# B&R Automation Studio project GroupProjectBR
Automation Studio 4.12.3.127 SP; Project that includes both HMI visualization and script of controling conveyor belt and sorting system.; technology packages: mapp 5.23.0, mappCockpit 5.23.0, mappMotion 5.23.0, mappView 5.23.0, mappVision 5.23.0

## Configuration ConfigSortingSystem

CPU , AutomationRuntime B4.93, Build 4.1.2, Safety 0.0, Vc V4.72.6

### Task classes (Cpu.sw)
```
Cyclic#4:
  Auto <- Programs.Auto.prg
  Camera <- Programs.Camera.prg
  Alarms <- Programs.Alarms.prg
  Manual <- Programs.Manual.prg
  ProgramRec <- Programs.RecipesMgmnt.prg
  SemiAuto <- Programs.SemiAuto.prg
DataObjects: McAcpSys
NcDataObjects: McDriveLog
Binaries: McAcpDrv, udbdef, McAcpSim, mvLoader, arflatprv, TCLang, visionUnit, mCoWebSc, TCData, FWRules, arcoal, arsvcreg, SettingsVi, sysconf, Settings, iomap, asfw, viComp, Role, ashwac, gRecipeXML, Config_2, arconfig, viAppLogo, Config_1, TC, ashwd, Config, User
Libraries: McBase, MpAxis, McAxis, MpBase, McAcpAx, CoTrace, AsZip, FileIO, runtime, ViBase, AsARCfg, powerlnk, MpRecipe, AsEPL, AsIO, DataObj, astime, MpAlarmX, MpServer, standard, AsHttp, asieccon, aruser, arssl, sys_lib, MpUserX
```

### Hardware
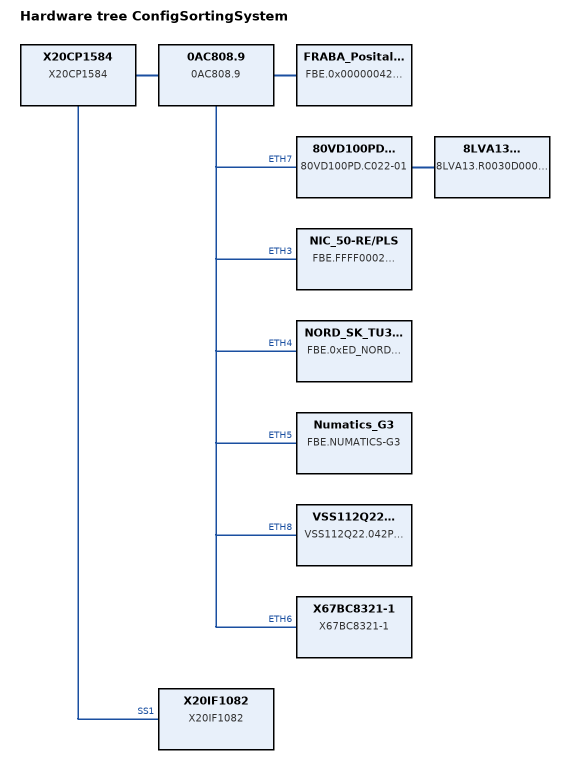
```
0AC808.9 : 0AC808.9 v1.0.0.0  [ETH1 -> X20CP1584.IF3 [Cable Type=PowerlinkCable, Length=10, Version=1.0.0.3]; ETH2 -> FRABA_Posital_Absolute_Rotary_Encoder.PLK1 [Cable Type=PowerlinkCable, Length=10, Version=1.0.0.3]; ETH3 -> NIC_50-RE/PLS.PLK1 [Cable Type=PowerlinkCable, Length=10, Version=1.0.0.3]; ETH4 -> NORD_SK_TU3-POL_SK54xE_Inverter.PLK1 [Cable Type=PowerlinkCable, Length=10, Version=1.0.0.3]; ETH5 -> Numatics_G3.PLK1 [Cable Type=PowerlinkCable, Length=10, Version=1.0.0.3]; ETH6 -> X67BC8321-1.PLK1 [Cable Type=PowerlinkCable, Length=10, Version=1.0.0.3]; ETH7 -> 80VD100PD.C022-01.PLK2 [Cable Type=PowerlinkCable, Length=10, Version=1.0.0.3]; ETH8 -> VSS112Q22.042P-000.PLK1 [Cable Type=PowerlinkCable, Length=10, Version=1.0.0.3]]
80VD100PD.C022-01 : 80VD100PD.C022-01 v2.5.0.0  [PLK2 -> 0AC808.9.ETH7 (NodeNumber=9) [Cable Type=PowerlinkCable, Length=10, Version=1.0.0.3]]
  DriveConfiguration/Module:
    McAcoposTypeID = AcoposMicroDConfig
    ActivateACOPOSSimulationOnPLC = 0
  DriveConfiguration/Encoder/EncoderX6A/InterfaceType:
    ResolverPolepairs = 1
  DriveConfiguration/Encoder/EncoderX6B/InterfaceType:
    ResolverPolepairs = 1
  DriveConfiguration/Channel[1]/RealAxis:
    AxisReference = gAxis_1
    MechanicalElementsIsInvisible = 0
  DriveConfiguration/Channel[1]/RealAxis/MechanicalElements/Gearbox:
    InputIsReadOnly = 0
    Input = 1
    OutputIsReadOnly = 0
    Output = 1
  DriveConfiguration/Channel[1]/RealAxis/MechanicalElements/RotaryToLinearTransformation:
    ReferenceDistanceIsReadOnly = 0
    ReferenceDistance = 175
  DriveConfiguration/Channel[1]/RealAxis/Controller:
    ModeIsReadOnly = 0
    Mode = PositionController
  DriveConfiguration/Channel[1]/RealAxis/Controller/Mode/Position:
    ProportionalGain = 194
    IntegrationTime = 0.0
    PredictionTime = 0.0004
    TotalDelayTime = 0.0004
  DriveConfiguration/Channel[1]/RealAxis/Controller/Mode/Speed:
    ProportionalGainIsReadOnly = 0
    ProportionalGain = 0.75
    IntegrationTimeIsReadOnly = 0
    IntegrationTime = 0.0
    FilterTimeIsReadOnly = 0
    FilterTime = 0.0
  DriveConfiguration/Channel[1]/RealAxis/Controller/Mode/LoopFilters:
    LoopFilterXIsReadOnly = 0
    LoopFilter1 = NotUsed
    LoopFilter2 = NotUsed
    LoopFilter3 = NotUsed
  DriveConfiguration/Channel[1]/RealAxis/Homing:
    ModeIsReadOnly = 0
    Mode = Direct
  DriveConfiguration/Channel[1]/RealAxis/Homing/Mode:
    Position = 0.0
    ReferencePulse = NotUsed
  DriveConfiguration/Channel[1]/RealAxis/Homing:
    RestorePositionVariable = 
  DriveConfiguration/Channel[1]/RealAxis/StopReaction:
    QuickstopIsReadOnly = 0
    Quickstop = DecelerationLimit
    DriveErrorIsReadOnly = 0
    DriveError = DecelerationLimit
  DriveConfiguration/Channel[1]/RealAxis/MovementErrorLimits:
    PositionError = 5
    VelocityErrorMonitoring = Automatic1
  DriveConfiguration/Channel[1]/RealAxis:
    JerkFilterIsReadOnly = 0
    JerkFilter = NotUsed
    ZeroVibrationFilter = NotUsed
  DriveConfiguration/Channel[1]/RealAxis/DigitalInputs/HomingSwitch:
    SourceIsReadOnly = 0
    Source = NotUsed
    Level = High
  DriveConfiguration/Channel[1]/RealAxis/DigitalInputs/PositiveLimitSwitch:
    SourceIsReadOnly = 0
    Source = NotUsed
    Level = High
  DriveConfiguration/Channel[1]/RealAxis/DigitalInputs/NegativeLimitSwitch:
    SourceIsReadOnly = 0
    Source = NotUsed
    Level = High
  DriveConfiguration/Channel[1]/RealAxis/DigitalInputs/Trigger1:
    Source = X2Trigger1
    Level = High
  DriveConfiguration/Channel[1]/RealAxis/DigitalInputs/Trigger2:
    Source = X2Trigger2
    Level = High
  DriveConfiguration/Channel[1]/RealAxis/DigitalInputs/Quickstop:
    Input = Trigger2
  DriveConfiguration/Channel[1]/RealAxis/Simulation:
    SimulationModeOnPLC = SetValueGeneration
    SimulationModeOnACOPOS = NotUsed
  DriveConfiguration/Channel[2]/RealAxis:
    AxisReference = 
    MechanicalElementsIsInvisible = 0
  DriveConfiguration/Channel[2]/RealAxis/MechanicalElements/Gearbox:
    InputIsReadOnly = 0
    Input = 1
    OutputIsReadOnly = 0
    Output = 1
  DriveConfiguration/Channel[2]/RealAxis/MechanicalElements/RotaryToLinearTransformation:
    ReferenceDistanceIsReadOnly = 0
    ReferenceDistance = 1
  DriveConfiguration/Channel[2]/RealAxis/Controller:
    ModeIsReadOnly = 0
    Mode = PositionController
  DriveConfiguration/Channel[2]/RealAxis/Controller/Mode/Position:
    ProportionalGain = 50.0
    IntegrationTime = 0.0
    PredictionTime = 0.0004
    TotalDelayTime = 0.0004
  DriveConfiguration/Channel[2]/RealAxis/Controller/Mode/Speed:
    ProportionalGainIsReadOnly = 0
    ProportionalGain = 2.0
    IntegrationTimeIsReadOnly = 0
    IntegrationTime = 0.0
    FilterTimeIsReadOnly = 0
    FilterTime = 0.0
  DriveConfiguration/Channel[2]/RealAxis/Controller/Mode/LoopFilters:
    LoopFilterXIsReadOnly = 0
    LoopFilter1 = NotUsed
    LoopFilter2 = NotUsed
    LoopFilter3 = NotUsed
  DriveConfiguration/Channel[2]/RealAxis/Homing:
    ModeIsReadOnly = 0
    Mode = Direct
  DriveConfiguration/Channel[2]/RealAxis/Homing/Mode:
    Position = 0.0
    ReferencePulse = NotUsed
  DriveConfiguration/Channel[2]/RealAxis/Homing:
    RestorePositionVariable = 
  DriveConfiguration/Channel[2]/RealAxis/StopReaction:
    QuickstopIsReadOnly = 0
    Quickstop = DecelerationLimit
    DriveErrorIsReadOnly = 0
    DriveError = DecelerationLimit
  DriveConfiguration/Channel[2]/RealAxis/MovementErrorLimits:
    PositionError = 1.0
    VelocityErrorMonitoring = Automatic1
  DriveConfiguration/Channel[2]/RealAxis:
    JerkFilterIsReadOnly = 0
    JerkFilter = NotUsed
    ZeroVibrationFilter = NotUsed
  DriveConfiguration/Channel[2]/RealAxis/DigitalInputs/HomingSwitch:
    SourceIsReadOnly = 0
    Source = NotUsed
    Level = High
  DriveConfiguration/Channel[2]/RealAxis/DigitalInputs/PositiveLimitSwitch:
    SourceIsReadOnly = 0
    Source = NotUsed
    Level = High
  DriveConfiguration/Channel[2]/RealAxis/DigitalInputs/NegativeLimitSwitch:
    SourceIsReadOnly = 0
    Source = NotUsed
    Level = High
  DriveConfiguration/Channel[2]/RealAxis/DigitalInputs/Trigger1:
    Source = X2Trigger1
    Level = High
  DriveConfiguration/Channel[2]/RealAxis/DigitalInputs/Trigger2:
    Source = X2Trigger2
    Level = High
  DriveConfiguration/Channel[2]/RealAxis/DigitalInputs/Quickstop:
    Input = Trigger2
  DriveConfiguration/Channel[2]/RealAxis/Simulation:
    SimulationModeOnPLC = SetValueGeneration
    SimulationModeOnACOPOS = NotUsed
8LVA13.R0030D000-0 : 8LVA13.R0030D000-0 v2.2.0.4  [MT -> 80VD100PD.C022-01.MT1]
  M1/MotorParameters:
    MOTOR_AMB_TEMP_RATED = 40
FRABA_Posital_Absolute_Rotary_Encoder : FBE.0x00000042_PowerlinkRotaryEncoder_OCD_V02-10 v1.0 (OrderNumber=FRABA Posital Absolute Rotary Encoder)  [PLK1 -> 0AC808.9.ETH2 (NodeNumber=8) [Cable Type=PowerlinkCable, Length=10, Version=1.0.0.3]]
  Supervision = off
  p2110_value = 
  p6000_value = 
  p6003_value = 
NIC_50-RE/PLS : FBE.FFFF0002_TLBPOWERLINK v1.0 (OrderNumber=NIC 50-RE/PLS)  [PLK1 -> 0AC808.9.ETH3 (NodeNumber=2) [Cable Type=PowerlinkCable, Length=10, Version=1.0.0.3]]
  Supervision = off
NORD_SK_TU3-POL_SK54xE_Inverter : FBE.0xED_NORD_TU3_POL_SK54xE_Inverter v1.0 (OrderNumber=NORD SK TU3-POL SK54xE Inverter)  [PLK1 -> 0AC808.9.ETH4 (NodeNumber=3) [Cable Type=PowerlinkCable, Length=10, Version=1.0.0.3]]
  Supervision = off
Numatics_G3 : FBE.NUMATICS-G3 v1.0 (OrderNumber=Numatics G3)  [PLK1 -> 0AC808.9.ETH5 (NodeNumber=6) [Cable Type=PowerlinkCable, Length=10, Version=1.0.0.3]]
  Supervision = off
VSS112Q22.042P-000 : VSS112Q22.042P-000 v1.7.0.605  [PLK1 -> 0AC808.9.ETH8 (NodeNumber=1) [Cable Type=PowerlinkCable, Length=10, Version=1.0.0.3]]
  Supervision = off
  VisionConfig = gCamera
X20CP1584 : X20CP1584 v1.10.0.0
  Connector IF2:
    ActivateDevice = 1
    Mode = Manual
    InternetAddress = 192.168.0.100
    SubnetMask = 255.255.255.0
    ActivateSnmp = 2
  Connector IF3:
    MtuSize = 1500
    CycleTime = 400
    InternetAddress = 192.168.200.240
    SubnetMask = 255.255.255.0
    ActivateANSL = 1
  ConfigurationID = Group_Project_BR_ConfigSortingSystem
  Simulation = 1
  TimerDeviceType = EPLX2X
  TimerDevice = X20CP1584.IF3
  TaskClassIdleTime = 2000
  FileDevice1
  FileDeviceName1 = CF
  FileDevicePath1 = C:\Users\Szkolenie\Desktop\Recipies
  FileDevice2
  FileDeviceName2 = TegesSmeges
  FileDevicePath2 = C:\Users\barto\OneDrive\Pulpit\Folder na receptury
  TimeZone = 160
  ActivateDaylightSavingTime = 1
  ActivateOpcUa = 1
  OpcUaInformationModels_PV_Version = 1
X20IF1082 : X20IF1082 v1.12.0.0  [SS -> X20CP1584.SS1]
  Connector IF1:
    EplNatSubnet = 192.168.102.0
X67BC8321-1 : X67BC8321-1 v2.14.0.0  [PLK1 -> 0AC808.9.ETH6 (NodeNumber=5) [Cable Type=PowerlinkCable, Length=10, Version=1.0.0.3]]
```

### IoMap.iom - X20CP1584/IoMap.iom
```iecst
VAR_CONFIG
	::gInWeightMeasure AT %IB."NIC_50-RE/PLS"._1ByteIn_04_I2100_S04;
	::Camera:PhotosTaken AT %IB."VSS112Q22.042P-000".CompletedAcquisitionCnt;
	::gActuatorByte AT %QW."Numatics_G3".Out01_I3201Out;
	::gImageAcq AT %QX."VSS112Q22.042P-000".ImageAcquisition;
	::Camera:SET_FOCUS AT %QW."VSS112Q22.042P-000".SetFocus;
	::Camera:EXPO_TIME AT %QD."VSS112Q22.042P-000".ExposureTime01;
	::Camera:NumberMatches AT %IB."VSS112Q22.042P-000".NumResultsMatch;
	::Camera:RecognisedModel AT %IB."VSS112Q22.042P-000".ModelNumberMatch01;
	::Camera:MatchEnable AT %QX."VSS112Q22.042P-000".EnableMatch;
	::Camera:NUM_SEARCH_MAX AT %QB."VSS112Q22.042P-000".NumSearchMaxMatch;
	::Camera:MIN_SCORE AT %QB."VSS112Q22.042P-000".MinScoreMatch;
	::Camera:MAX_OVERLAP AT %QB."VSS112Q22.042P-000".MaxOverlapMatch;
	::Camera:FLASH_COLOR AT %QB."VSS112Q22.042P-000".FlashColor01;
	::Camera:FLASH_SEGMENT AT %QB."VSS112Q22.042P-000".FlashSegment01;
	::Camera:MatchScore AT %IB."VSS112Q22.042P-000".ScoreMatch01;
	::Camera:CameraLED_OPC AT %QB."VSS112Q22.042P-000".StatusLED;
	::Camera:ImgProcessingActive AT %IX."VSS112Q22.042P-000".ImageProcessingActive;
	::Alarms:ModuleOkCamera AT %IX."VSS112Q22.042P-000".ModuleOk;
	::Alarms:ModuleOkScale AT %IX."NIC_50-RE/PLS".ModuleOk;
	::Alarms:ModuleOkInverter AT %IX."NORD_SK_TU3-POL_SK54xE_Inverter".ModuleOk;
	::Alarms:ModuleOkPLC_PLK AT %IX."X20IF1082".ModuleOk;
	::Alarms:ModuleOkEncoder AT %IX."FRABA_Posital_Absolute_Rotary_Encoder".ModuleOk;
	::Alarms:ModuleOkActuators AT %IX."Numatics_G3".ModuleOk;
	::Alarms:ModuleOkPneu_X67BC AT %IX."X67BC8321-1".ModuleOk;
END_VAR
```

### Config.mpalarmxcore - X20CP1584/mappServices/Config.mpalarmxcore
```
Element gAlarmXCore (Type=mpalarmxcore)
  mapp.AlarmX.Core.Configuration:
    [0]:
      Name = Unrecognized object
      Message = Attempt to classify object has failed
      Behavior = DiscreteValueMonitoring
        Monitoring:
          MonitoredPV = ::Auto:State
          TriggerValues:
            [0] = 14
    [1]:
      Name = Left box is full
      Message = Left box reached maximum ammount of objects in it
      Behavior = LevelMonitoring
        Monitoring:
          MonitoredPV = ::Auto:QuantityLeftStorage
          HighLimitEnable = Dynamic
            LimitPV = ::gMaxLeftStorage
    [2]:
      Name = Right box is full
      Message = Right box reached maximum ammount of objects in it
      Behavior = LevelMonitoring
        Monitoring:
          MonitoredPV = ::Auto:QuantityRightStorage
          HighLimitEnable = Dynamic
            LimitPV = ::gMaxRightStorage
    [3]:
      Name = Motor error
      Message = gMotorBeltAxisBasic has returned an error. Manual restart is required in "Service" page.
      Behavior = DiscreteValueMonitoring
        Monitoring:
          MonitoredPV = ::gMotorBeltAxisBasic.Error
          TriggerValues:
            [0] = 1
    [4]:
      Name = Right box is full (manual)
      Message = Right box reached maximum ammount of objects in it (manual mode)
      Behavior = LevelMonitoring
        Monitoring:
          MonitoredPV = ::SemiAuto:QuantityRightStorage
          HighLimitEnable = Dynamic
            LimitPV = ::gMaxRightStorage
    [5]:
      Name = Left box is full (manual)
      Message = Left box reached maximum ammount of objects in it (manual mode)
      Behavior = LevelMonitoring
        Monitoring:
          MonitoredPV = ::SemiAuto:QuantityLeftStorage
          HighLimitEnable = Dynamic
            LimitPV = ::gMaxRightStorage
    [6]:
      Name = Hardware error
      Message = No connection to at least on module. Fix connections and reset hardware via service page
      Behavior = DiscreteValueMonitoring
        Monitoring:
          MonitoredPV = ::gAlarmHardware
          TriggerValues:
            [0] = 1
```

### viComp.visioncomponent - X20CP1584/mappVision/viComp.visioncomponent
```
Element gCamera (Type=visioncomponent)
  VisionApplicationReference = viAppLogo
```

## Logical view

Binary libraries used (declarations not repeated): operator, runtime, astime, AsIecCon, MpAxis, McAxis, MpBase, McAcpAx, CoTrace, AsZip, FileIO, McBase, MpRecipe, asstring, ViBase, AsARCfg, powerlnk, AsEPL, AsIO, DataObj, MpAlarmX, MpServer, standard, AsHttp

### Global.typ - Global data types
```iecst
TYPE
	ModelEnum :
		(
		BR := 1, (*%ID of B&R logo model*)
		AS := 2, (*%ID of AS logo model*)
		Unrecognised := 0 (*%case of nothing recognised*)
		);
	CofeeType : 	STRUCT
		Sugar : USINT;
		Water : REAL;
		Powder : USINT;
		Temperature : REAL;
		Milk : REAL;
	END_STRUCT;
	SortingType : 	STRUCT
		RecognisedModel : ModelEnum; (*Model rozpoznany*)
		ItemWeightChoosen : USINT := 10;
		SortLeftMin : BOOL := FALSE; (*Mniejsze detale sortowane są na lewo gdy 1, a wieksze na prawo gdy 1.*)
		SortLeftBR : BOOL := FALSE; (*Gdy ustawiona na 1 sortuje BR na lewo, a AS na prawo*)
		SortChoice : SortChoiceEnum;
	END_STRUCT;
	SortChoiceEnum :
		(
		WEIGHT,
		OPTIC
		);
END_TYPE
```

### Global.var - Global variables
```iecst
(*Insert your comment here.*)
VAR
	Coffee : CofeeType;
	gActuatorByte : UINT;
	gAlarmExist : BOOL := FALSE;
	gAlarmHardAck : BOOL := FALSE;
	gAlarmHardware : BOOL := FALSE;
	gAutoRecipe : USINT;
	gErrorState : BOOL := FALSE;
	gExposureTime : UDINT;
	gImageAcq : BOOL := FALSE; (*Enabling image acquisition therefore starting matching procedure, rising edge*)
	gInWeightMeasure : USINT;
	gItemWeightChoosen : USINT := 10;
	gMaxLeftStorage : USINT := 4;
	gMaxRightStorage : USINT := 4;
	gMode : USINT := 0;
	gMotorBeltAxisBasic : MpAxisBasic;
	gMotorBeltParType : MpAxisBasicParType;
	gMpRecipeRegPar_0 : MpRecipeRegPar;
	gMpRecipeUI_0 : MpRecipeUI;
	gMpRecipeXML_0 : MpRecipeXml;
	gPicNotRecognised : BOOL := FALSE;
	gRecognisedModel : ModelEnum := Unrecognised; (*Value showing recognised model 1- B&R, 2- AS, 0- not recognised*)
	gSetFocus : USINT;
	gSortChoice : SortChoiceEnum := WEIGHT;
	gSortChoiceView : BOOL;
	gSorting : SortingType;
	gStopBlink : BOOL := TRUE;
	gStopState : BOOL := TRUE;
	gUIConnect : MpRecipeUIConnectType;
	gUISetup : MpRecipeUISetupType;
	gWeightDetected : BOOL := FALSE;
	gDisplayImg : BOOL;
END_VAR
```

### Package Logical/Libraries - Global libraries

- Visualisation Logical/mappView (not shown)

### Program Logical/Programs/Auto (IEC)

#### Types.typ
```iecst
TYPE
	ProgramStatesEnum :
		(
		STOP,
		INIT,
		DETECTION,
		CATEGORIZATION,
		SORT_STORAGE_LEFT,
		SORT_STORAGE_RIGHT,
		SORT_WEIGHT,
		SORT_WEIGHT_AND_OPTIC,
		SORT_OPTIC,
		STOP_AND_MANUAL,
		GO_STORAGE_LEFT,
		GO_STORAGE_RIGHT,
		TAKE_PICT_CAMERA,
		DROP,
		UNRECOGNISED_PIC,
		ERROR
		);
END_TYPE
```

#### Variables.var
```iecst
VAR
	TIME_TON_DETECT : TIME := T#2S;
END_VAR
VAR CONSTANT
	TIME_TON_CAMERA : TIME := T#4S;
	TIME_TON_ACTUATOR : TIME := T#500MS;
END_VAR
VAR
	TimerTonDetect : TON;
	TimerTonCamera : TON;
	TimerTonActuatorIn : BOOL := FALSE;
	TimerTonActuator : TON;
	TimerCameraPicDone : BOOL;
	TimerAfterDetect : BOOL;
	TimerActuatorOut : BOOL;
	StringState : STRING[80];
	StringRecognisedModel : STRING[80];
	Stop : BOOL := FALSE;
	State : ProgramStatesEnum := STOP;
	Start : BOOL := FALSE;
	SelectedAuto : BOOL;
	RESET_ITEM_MEM_WEIGHT : {REDUND_UNREPLICABLE} USINT := 0;
	NotSelectedAuto : BOOL;
END_VAR
VAR CONSTANT
	MOTOR_DIST_RIGHT : UINT := 320;
	MOTOR_DIST_LEFT : UINT := 90;
END_VAR
VAR
	MotorVel : REAL;
	MotorResetError : BOOL := FALSE;
	MotorReqVel : {REDUND_UNREPLICABLE} UINT := 300;
	MotorReqPosition : UINT := 0;
	MotorReqDec : UINT := 700;
	MotorReqAcc : UINT := 700;
	MotorPower : BOOL := FALSE;
	MotorPos : LREAL;
	MotorMoveDone : BOOL;
	MotorMoveAbsolute : BOOL := FALSE;
	MotorInPosition : BOOL;
	MotorHome : BOOL;
	ItemWeightMeasured : USINT;
	ItemWeight : USINT;
	ItemDetected : BOOL := FALSE;
	IsEnglishSelected : BOOL := TRUE;
END_VAR
VAR CONSTANT
	ACTUATOR_BYTE_SORT : INT := 2#0000000000000001;
	ACTUATOR_BYTE_PUSH : INT := 2#0000000000000100;
	ACTUATOR_BYTE_NOT_ACTIV : USINT := 2#0000000000000000;
END_VAR
VAR
	ActuatorSorting : BOOL := FALSE;
	ActuatorPushing : BOOL := FALSE;
	ActuatorNotSorting : BOOL;
	ActuatorNotPushing : BOOL;
	ActuatorByte : INT := 2#0000000000000000;
END_VAR
```

#### Main.st
```iecst
PROGRAM _INIT
	// NEED ONLY FOR WATCH
	gAxis_1;
	gMotorBeltParType;
	gMotorBeltAxisBasic;
END_PROGRAM
//po namyśle można było użyć struktur do zmiennych :P
PROGRAM _CYCLIC

	SelectedAuto := (gMode = 0);
	NotSelectedAuto := NOT SelectedAuto;

	// CODE WORKS ONLY WHEN AUTO IS ACTIVE
	IF  SelectedAuto THEN
		// MOTOR MANAGEMENT
		gMotorBeltAxisBasic.Enable 		:= TRUE;
		gMotorBeltAxisBasic.MpLink 		:= ADR(gAxis_1);
		gMotorBeltAxisBasic.Parameters 	:= ADR(gMotorBeltParType);
		MotorMoveDone 					:= gMotorBeltAxisBasic.MoveDone;
		gMotorBeltAxisBasic.Power 		:= MotorPower;
		gMotorBeltAxisBasic.Home 		:= MotorHome;

		gMotorBeltAxisBasic();

		// IN STATE STOP VALUES DOESN'T FLUCTUATE
		IF gMotorBeltAxisBasic.Velocity > 15 THEN
			MotorVel := gMotorBeltAxisBasic.Velocity;
		ELSE
			MotorVel := 0;
		END_IF;
		IF gMotorBeltAxisBasic.Position > 5 THEN
			MotorPos := gMotorBeltAxisBasic.Position;
		ELSE
			MotorPos := 0;
		END_IF;

		// ASSIGNING MOTION PARAMETERS
		gMotorBeltParType.Acceleration 	:= MotorReqAcc;
		gMotorBeltParType.Deceleration 	:= MotorReqDec;
		gMotorBeltParType.Velocity 		:= MotorReqVel;
		gMotorBeltParType.Position 		:= MotorReqPosition;

		// ASSIGNING GLOBAL VARIABLES TO LOCAL VARIABLES
		gActuatorByte					 := ActuatorByte;
		gMotorBeltAxisBasic.Power 		 := MotorPower;
		gMotorBeltAxisBasic.MoveAbsolute := MotorMoveAbsolute;
		gStopState 						 := (State = 0);

		// ASSIGNING LOCAL VARIABLES TO GLOBAL VARIABLES
		MotorInPosition 				 := gMotorBeltAxisBasic.InPosition;
		ItemWeight 						 := gInWeightMeasure;

		// ITEM DETECTION CONDITION
		ItemDetected := (ItemWeight > 1);
		gWeightDetected := ItemDetected;

		// TIMERS
		// actuator
		TimerTonActuator(IN := TimerTonActuatorIn, PT := TIME_TON_ACTUATOR);
		TimerActuatorOut := TimerTonActuator.Q;
		// camera
		TimerTonCamera(IN := gImageAcq , PT := TIME_TON_CAMERA);
		TimerCameraPicDone := TimerTonCamera.Q;
		// delay after detection
		TimerTonDetect.IN := ItemDetected;
		TimerTonDetect.PT := TIME_TON_DETECT;
		TimerAfterDetect := TimerTonDetect.Q;
		TimerTonDetect();

	END_IF;

	// ALARM OR STOP OR AUTO NOT ACTIVE
	IF	gAlarmHardware THEN
		IF NOT (State = ERROR) THEN
			State := ERROR;
		END_IF;
	ELSIF Stop OR gMode <> 0 OR gAlarmExist THEN
		Stop := FALSE;
		State := STOP;
	END_IF;

	// PROGRAM AUTO
	CASE State OF
		STOP:
			IF SelectedAuto THEN
				MotorPower 		  := FALSE;
				MotorMoveAbsolute := FALSE;
				MotorHome 		  := FALSE;
			END_IF;
			MotorPos := 0;
			MotorVel := 0;
			StringState := 'Stop';
			TimerTonActuatorIn 	  := FALSE;
			ActuatorSorting 	  := FALSE;
			ActuatorPushing  	  := FALSE;
			IF Start THEN
				State := INIT;
			END_IF;

		INIT:
			StringState 		:= 'Inicjalizacja';
			gAddToRight 		:= FALSE;
			gAddToLeft 			:= FALSE;
			TimerTonActuatorIn 	:= FALSE;
			ActuatorSorting 	:= FALSE;
			ActuatorPushing 	:= FALSE;
			MotorMoveAbsolute 	:= FALSE;
			MotorPower 			:= TRUE;
			MotorHome 			:= TRUE;
			gPicNotRecognised	:= FALSE;
			State 				:= START;

		START:
			StringState 		:= 'Gotowy do startu';
			IF ItemDetected THEN
				ItemWeightMeasured 	:= RESET_ITEM_MEM_WEIGHT;
				State := DETECTION;
			END_IF;

		DETECTION:
			MotorHome 	:= FALSE;
			StringState := 'Wykrycie detalu';
			IF TimerAfterDetect THEN
				ItemWeightMeasured := ItemWeight;
				State := CATEGORIZATION;
			END_IF;

		CATEGORIZATION:
			StringState := 'Kategoryzacja detalu';
			IF gSorting.SortChoice = WEIGHT THEN
				State := DROP;
			ELSIF gSorting.SortChoice = OPTIC THEN
				State := TAKE_PICT_CAMERA;
			END_IF;

		TAKE_PICT_CAMERA:
			StringState := 'Robienie zdjecia';
			gImageAcq 	:= TRUE;
			IF TimerCameraPicDone THEN
				gDisplayImg := TRUE;
				IF gSorting.RecognisedModel = 0 THEN 						//0
					gImageAcq 			  := FALSE;
					StringRecognisedModel := 'Unrecognised';
					State 				  := UNRECOGNISED_PIC;
				ELSE
					State 				  := DROP;
				END_IF;
			END_IF;

		DROP:
			StringState := 'Dozowanie detalu';
			ActuatorPushing := TRUE;
			IF TimerActuatorOut THEN
				ActuatorPushing := FALSE;
				IF gSorting.SortChoice = OPTIC THEN
					gSortChoiceView := TRUE;
					State := SORT_OPTIC;
				ELSIF gSorting.SortChoice = WEIGHT THEN
					gSortChoiceView := FALSE;
					State := SORT_WEIGHT;
				END_IF;
			END_IF;

			// ABOVE 1 TO ItemWeightChoosen ITEM FALL INTO THE LEFT, EQUAL AND ABOVE ItemWeightChoosen INTO THE RIGHT
		SORT_WEIGHT:
			StringState := 'Sortowanie wagowe';
			IF ItemWeightMeasured > 1 AND ItemWeightMeasured < gSorting.ItemWeightChoosen THEN
				IF gSorting.SortLeftMin THEN
					State := GO_STORAGE_LEFT;
				ELSE
					State := GO_STORAGE_RIGHT;
				END_IF;
			ELSIF ItemWeightMeasured >= gSorting.ItemWeightChoosen THEN
				IF gSorting.SortLeftMin THEN
					State := GO_STORAGE_RIGHT;
				ELSE
					State := GO_STORAGE_LEFT;
				END_IF;
			END_IF;

		SORT_OPTIC:
			StringState := 'Sortowanie optyczne';
			IF gSorting.RecognisedModel = 1 THEN
				gImageAcq 			  := FALSE;
				StringRecognisedModel := 'B&R';							//1
				IF gSorting.SortLeftBR THEN
					State := GO_STORAGE_LEFT;
				ELSE
					State := GO_STORAGE_RIGHT;
				END_IF;

			ELSIF gSorting.RecognisedModel = 2 THEN
				gImageAcq 			  := FALSE;
				StringRecognisedModel := 'AS';							//2
				IF gSorting.SortLeftBR THEN
					State := GO_STORAGE_RIGHT;
				ELSE
					State := GO_STORAGE_LEFT;
				END_IF;
			END_IF;

		GO_STORAGE_LEFT:
			StringState := 'Transport detalu do lewego zbiornika';
			MotorReqPosition := MOTOR_DIST_LEFT;
			MotorMoveAbsolute := TRUE;
			IF MotorInPosition AND MotorMoveDone THEN
				State := SORT_STORAGE_LEFT;
			END_IF;

		GO_STORAGE_RIGHT:
			StringState := 'Transport detalu do prawego zbiornika';
			MotorReqPosition  := MOTOR_DIST_RIGHT;
			MotorMoveAbsolute := TRUE;
			IF MotorInPosition AND MotorMoveDone THEN
				State := SORT_STORAGE_RIGHT;
			END_IF;

		SORT_STORAGE_LEFT:
			StringState := 'Zepchniecie detalu z tasmy do zbiornika lewego';
			MotorMoveAbsolute := FALSE;
			ActuatorSorting   := TRUE;
			gAddToLeft 		  := TRUE;
			IF TimerActuatorOut THEN
				State := INIT;
			END_IF;

		SORT_STORAGE_RIGHT:
			gAddToRight := TRUE;
			MotorMoveAbsolute := FALSE;
			State := INIT;

		UNRECOGNISED_PIC:
			StringState := 'Nie rozpoznano zdjecia';
			gPicNotRecognised := TRUE;
			State := STOP;

		ERROR: // SPONTANICZNA DECYZJA CTRL V Z STOP DLA LEPSZEJ FUNKCJONALNOŚCI - BRAKLO CZASU NA DOKLADNIEJSZE POPRAWKI
			IF gMode = 0 THEN
				MotorPower 		  := FALSE;
				MotorMoveAbsolute := FALSE;
				MotorHome 		  := FALSE;
			END_IF;
			MotorPos := 0;
			MotorVel := 0;
			TimerTonActuatorIn 	  := FALSE;
			ActuatorSorting 	  := FALSE;
			ActuatorPushing  	  := FALSE;
			StringState := 'Wystapil blad';
			gErrorState := TRUE;
			IF gAlarmHardAck THEN
				IF NOT gAlarmHardware THEN
					gAlarmHardAck := FALSE;
					gErrorState := FALSE;
					State := STOP;
				END_IF;
			END_IF;

	END_CASE;

	// TIMER INPUT TRIGGER TO DELAY ACTUATORS
	IF ActuatorPushing OR ActuatorSorting THEN
		TimerTonActuatorIn := TRUE;
	ELSE
		TimerTonActuatorIn := FALSE;
	END_IF;

	// OPERATION OF BYTE ACTUATORS WITH TIMER
	IF ActuatorPushing THEN
		ActuatorByte := ACTUATOR_BYTE_PUSH;
		IF TimerActuatorOut THEN
			ActuatorPushing := FALSE;
		END_IF;
	ELSIF ActuatorSorting THEN
		ActuatorByte := ACTUATOR_BYTE_SORT;
		IF TimerActuatorOut THEN
			ActuatorSorting := FALSE;
		END_IF;
	ELSE
		ActuatorByte := ACTUATOR_BYTE_NOT_ACTIV;
	END_IF;

	// COUNTERS
	gCTU_QuantityLeft(CU := gAddToLeft, RESET := gCTU_Reset_Left, PV := gMaxLeftStorage);
	gCTU_QuantityRight(CU := gAddToRight, RESET := gCTU_Reset_Right, PV := gMaxRightStorage);
	gQuantityLeftStorage  := gCTU_QuantityLeft.CV;
	gQuantityRightStorage := gCTU_QuantityRight.CV;

	gCTU_QuantityLeft();
	gCTU_QuantityRight();

	// HMI GUYS WANTED SOME VARIABLES
	IF gSorting.SortChoice = OPTIC THEN
		gSortChoiceView := TRUE;
	ELSIF gSorting.SortChoice = WEIGHT THEN
		gSortChoiceView := FALSE;
	END_IF;

	ActuatorNotSorting := NOT ActuatorSorting;
	ActuatorNotPushing 	:= NOT ActuatorPushing;

	IF Start THEN
		Start := FALSE;
	END_IF;

	//Added by Jakub; Responsibler for changing machine state between English and Polish
	IF IsEnglishSelected THEN
		IF StringState = 'Inicjalizacja' THEN
			StringState := 'Initialization';

		ELSIF StringState = 'Gotowy do startu' THEN
			StringState := 'Ready';

		ELSIF StringState = 'Wykrycie detalu' THEN
			StringState := 'Item detection';

		ELSIF StringState = 'Kategoryzacja detalu' THEN
			StringState := 'Item categorization';

		ELSIF StringState = 'Robienie zdjecia' THEN
			StringState := 'Taking a picture';

		ELSIF StringState = 'Dozowanie detalu' THEN
			StringState := 'Item dosing';

		ELSIF StringState = 'Sortowanie wagowe' THEN
			StringState := 'Sorting by weight';

		ELSIF StringState = 'Sortowanie optyczne' THEN
			StringState := 'Optical sorting';

		ELSIF StringState = 'Transport detalu do lewego zbiornika' THEN
			StringState := 'Item transport to the left tank';

		ELSIF StringState = 'Transport detalu do prawego zbiornika' THEN
			StringState := 'Item transport to the right tank';

		ELSIF StringState = 'Zepchniecie detalu z tasmy do zbiornika lewego' THEN
			StringState := 'Pushing the item from the belt to the left tank';

		ELSIF StringState = 'Nie rozpoznano zdjecia' THEN
			StringState := 'Photo not recognized';

		ELSIF StringState = 'Stop' THEN
			StringState := 'Stop';

		ELSIF StringState = 'Wystapil blad' THEN
			StringState := 'Error';

		ELSIF StringState = 'Gotowy do startu' THEN
			StringState := 'Ready to start';
		END_IF;
	END_IF;

		END_PROGRAM

PROGRAM _EXIT

		END_PROGRAM
```

### Program Logical/Programs/Manual (IEC)

#### Types.typ
```iecst
TYPE
	AxisParam : 	STRUCT
		ManualDistance : LREAL := 500; (*Setting distance of the belt move [mm]*)
		ManualVelocity : REAL := 50; (*Value of velocity [mm/s]*)
	END_STRUCT;
	ManualStepsEnum :
		(
		MANUAL_WAIT := 10,
		MANUAL_BELT_SET_ADDITIVE := 20,
		MANUAL_BELT_MOVE_ADDITIVE := 30,
		MANUAL_BELT_SET_VELOCITY := 40,
		MANUAL_BELT_MOVE_VELOCITY := 50,
		MANUAL_BELT_MOVE_ADDITIVE1 := 60
		);
	ManualStepsActEnum :
		(
		MANUAL_ACTUATOR_WAIT := 200,
		MANUAL_ACTUATOR_DOSING := 210,
		MANUAL_ACTUATOR_NONE := 220,
		MANUAL_ACTUATOR_BOTH := 230,
		MANUAL_ACTUATOR_SORTING := 240
		);
END_TYPE
```

#### Variables.var
```iecst
VAR
	JogEnableVar : BOOL; (*Jog enablling variable*)
	FlagAdd : BOOL; (*Flag that enables user to see if additive move is active*)
	ManualStep : ManualStepsEnum; (*Enum steps of Manual's state machine*)
	ManualStop : BOOL := FALSE; (*Stopping all of the processes*)
	ManualDistance : LREAL := 300; (*Setting distance of the belt move [mm]*)
	ManualActuatorDosing : BOOL; (*Enabling dosing actuator*)
	ManualActuatorSorting : BOOL; (*Enabling sorting actuator*)
	ManualActuatorBoth : BOOL; (*Enabling both actuators*)
	BeltMoveAdditive : BOOL; (*Activating additive move*)
	ManualActuatorNone : BOOL; (*Disabling both actuators*)
	BeltMoveVelocityOn : BOOL; (*Activating velocity move*)
	BeltMoveVelocityOff : BOOL; (*Disactivating velocity move*)
	ManualVelocity : REAL := 50; (*Value of velocity [mm/s]*)
	StartButtonState : BOOL; (*State of Manual Start button*)
	DirectionChangeVelocity : BOOL; (*Switching the direction of velocity value / multiplying by -1*)
	DirectionChangeDistance : BOOL; (*Switching the direction of distance value / multiplying by -1*)
	FlagActBoth : BOOL; (*Flag for both enabled actuators*)
	FlagActNone : BOOL; (*Flag for none of enabled actuators*)
	FlagActSorting : BOOL; (*Flag for sorting actuator enabled *)
	FlagActDosing : BOOL; (*Flag for dosing actuator enabled*)
	MC_BR_JogVelocity_0 : MC_BR_JogVelocity; (*Jog velocity*)
	FlagManual : BOOL; (*Flag that enables user to see if manual mode is enabled*)
	ExposureTime : UDINT; (*Camera exposure time*)
	SetFocus : USINT; (*Setting focus of camera*)
	ManualStepAct : ManualStepsActEnum; (*Steps of the actuator state machine*)
	FlagActBothOff : BOOL; (*Flag of the disabled both of actuators*)
	FlagActDosingOff : BOOL; (*Flag of the disabled dosing actuator*)
	FlagActNoneOff : BOOL; (*Flag of the disabled both of actuators*)
	FlagActSortingOff : BOOL; (*Flag of the disabled sorting actuator*)
	FlagNotManual : BOOL; (*Flag that enables user to see if manual mode is disabled*)
	NotMoveActive : BOOL; (*Flag that enables user to see if move is not active*)
	AxisPowerOn : BOOL; (*Enabling power of the motor*)
	FlagArrowLeft : BOOL; (*Motor is rotating to the left side*)
	FlagArrowRight : BOOL; (*Motor is rotating to the right side*)
	AxisPowerOff : BOOL; (*Turning off the power of the axis*)
	FlagVelAddOff : BOOL; (*Flag that enables user to see if additive and velocity move is turned off*)
	PhotoShoot : BOOL; (*Shooting a photo*)
	PhotoShow : BOOL; (*Displaying a photo*)
	FlagVel : BOOL; (*Flag that enables user to see if velocity  move is active*)
	sCamera : USINT;
	ImageTON : TON;
END_VAR
```

#### Main.st
```iecst
PROGRAM _INIT

END_PROGRAM

PROGRAM _CYCLIC

	gMotorBeltAxisBasic();

	gAxis_1;

	gExposureTime;
	gSetFocus;

	NotMoveActive := NOT(gMotorBeltAxisBasic.MoveActive);

	IF PhotoShoot THEN
		PhotoShoot :=0;
	END_IF;

	IF PhotoShow THEN
		gDisplayImg := 1;
	ELSE
		gDisplayImg := 0;
	END_IF;

	//--------------DIRECTION---CHANGES--------------//
	IF DirectionChangeVelocity THEN
		DirectionChangeVelocity := 0;
		ManualVelocity := (-1)*ManualVelocity;
	END_IF;

	IF DirectionChangeDistance THEN
		DirectionChangeDistance := 0;
		ManualDistance := (-1)*ManualDistance;
	END_IF;

	//---------AXIS---VARIABLES---ASSIGMENT----------//

	IF gMode = 1 THEN
		gMotorBeltParType.Distance := ManualDistance;
		gMotorBeltParType.Velocity := ManualVelocity;
	END_IF;

	//-----------------MANUAL---STOP-----------------//
	IF ManualStop THEN
		ManualStop := 0;
		gActuatorByte := 2#0000_0000_0000_0000;
		gMotorBeltAxisBasic.MoveVelocity := 0;
		gMotorBeltAxisBasic.MoveAdditive := 0;
		gMotorBeltAxisBasic.Home := 0;
		gMotorBeltAxisBasic.Power := 0;
		ManualStep := MANUAL_WAIT;
		ManualStepAct := MANUAL_ACTUATOR_WAIT;
	END_IF;

	FlagVelAddOff;

	//----------------------MANUAL---MODE---CHECK---CONDITION----------------------//
	IF (gMode = 1) THEN

		//----------------------STATE---MACHINE---AXIS------------------------//
		CASE ManualStep OF

			MANUAL_WAIT:
				FlagVelAddOff := 1;
				FlagAdd := 0;
				FlagVel := 0;
				IF BeltMoveAdditive THEN
					gMotorBeltAxisBasic.Home := 0;
					BeltMoveAdditive := 0;
					FlagVelAddOff := 0;
					FlagAdd := 1;
					ManualStep := MANUAL_BELT_SET_ADDITIVE;
				ELSIF BeltMoveVelocityOn THEN
					gMotorBeltAxisBasic.Home := 0;
					BeltMoveVelocityOn := 0;
					FlagVelAddOff := 0;
					FlagVel := 1;
					ManualStep := MANUAL_BELT_SET_VELOCITY;
				END_IF;

			MANUAL_BELT_SET_ADDITIVE:
				ManualVelocity := ABS(ManualVelocity);
				gMotorBeltAxisBasic.Power := 0;
				gMotorBeltAxisBasic.Power := 1;
				IF gMotorBeltAxisBasic.PowerOn THEN
					gMotorBeltAxisBasic.Home := 0;
					ManualStep := MANUAL_BELT_MOVE_ADDITIVE;
				END_IF;

			MANUAL_BELT_MOVE_ADDITIVE:
				gMotorBeltAxisBasic.MoveAdditive := 1;
				IF gMotorBeltAxisBasic.MoveDone THEN
					gMotorBeltAxisBasic.ErrorReset := 1;
					gMotorBeltAxisBasic.MoveAdditive := 0;
					ManualStep := MANUAL_BELT_MOVE_ADDITIVE1;
				END_IF;

			MANUAL_BELT_MOVE_ADDITIVE1:
				gMotorBeltAxisBasic.ErrorReset := 0;
				ManualStep := MANUAL_WAIT;

			MANUAL_BELT_SET_VELOCITY:
				gMotorBeltAxisBasic.Power := 0;
				gMotorBeltAxisBasic.Power := 1;
				IF gMotorBeltAxisBasic.PowerOn THEN
					gMotorBeltAxisBasic.MoveVelocity := 1;
					ManualStep := MANUAL_BELT_MOVE_VELOCITY;
				END_IF;

			MANUAL_BELT_MOVE_VELOCITY:
				IF gMotorBeltAxisBasic.InVelocity THEN
					IF BeltMoveVelocityOff THEN
						BeltMoveVelocityOff := 0;
						gMotorBeltAxisBasic.MoveVelocity := 0;
						ManualStep := MANUAL_WAIT;
					END_IF;
				END_IF;
		END_CASE;

		//-------------------STATE---MACHINE---ACTUATORS---------------------//
		CASE ManualStepAct OF
			MANUAL_ACTUATOR_WAIT:
				IF ManualActuatorDosing THEN
					ManualActuatorDosing := 0;
					ManualStepAct := MANUAL_ACTUATOR_DOSING;
				ELSIF ManualActuatorSorting THEN
					ManualActuatorSorting := 0;
					ManualStepAct := MANUAL_ACTUATOR_SORTING;
				ELSIF ManualActuatorBoth THEN
					ManualActuatorBoth := 0;
					ManualStepAct := MANUAL_ACTUATOR_BOTH;
				ELSIF ManualActuatorNone THEN
					ManualActuatorNone := 0;
					ManualStepAct := MANUAL_ACTUATOR_NONE;
				END_IF;

			MANUAL_ACTUATOR_DOSING:
				gActuatorByte := 2#0000_0000_0000_0000;
				gActuatorByte := 2#0000_0000_0000_0100;
				ManualStepAct := MANUAL_ACTUATOR_WAIT;

				//actuating actuator responsibile for sorting an element
			MANUAL_ACTUATOR_SORTING:
				gActuatorByte := 2#0000_0000_0000_0000;
				gActuatorByte := 2#0000_0000_0000_0001;
				ManualStepAct := MANUAL_ACTUATOR_WAIT;

				//actuating both actuators
			MANUAL_ACTUATOR_BOTH:
				gActuatorByte := 2#0000_0000_0000_0000;
				gActuatorByte := 2#0000_0000_0000_0101;
				ManualStepAct := MANUAL_ACTUATOR_WAIT;

				//disactuating both actuators
			MANUAL_ACTUATOR_NONE:
				gActuatorByte := 2#0000_0000_0000_0000;
				ManualStepAct := MANUAL_ACTUATOR_WAIT;
		END_CASE;

		//------------END---OF---STATE---MACHINE---ACTUATORS---------------//
		IF AxisPowerOn THEN
			AxisPowerOn := 0;
			gMotorBeltAxisBasic.Power :=1;	//Axis power off is enabling by the button that is binded with stop step
		END_IF;
	END_IF;

	//----------------------------FLAG---SECTION----------------------------//
	IF (FlagActDosing = FALSE AND FlagActDosingOff = FALSE) THEN
		FlagActDosingOff := TRUE;
	END_IF;
	IF (FlagActSorting = FALSE AND FlagActSortingOff = FALSE) THEN
		FlagActSortingOff := TRUE;
	END_IF;

	//strzalka
	//robienie zdjecia

	//	IF ((ManualStep = MANUAL_BELT_SET_ADDITIVE) OR (ManualStep = MANUAL_BELT_MOVE_ADDITIVE)) AND  THEN
	//
	//	ELSIF ManualStep =
	//
	//	END_IF;

	IF gMotorBeltAxisBasic.PowerOn THEN
		AxisPowerOff := 1;
	ELSE
		AxisPowerOff := 0;
	END_IF;

	IF gMode = 1 THEN
		FlagManual := 1;
		FlagNotManual := 0;
	ELSE
		FlagNotManual := 1;
		FlagManual := 0;
	END_IF;

	IF ManualStepAct = MANUAL_ACTUATOR_DOSING THEN
		FlagActBoth := 0;
		FlagActBothOff := NOT(FlagActBoth);
		FlagActDosing := 1;
		FlagActDosingOff := NOT(FlagActDosing);
		FlagActNone := 0;
		FlagActNoneOff := NOT(FlagActNone);
		FlagActSorting := 0;
		FlagActSortingOff := NOT(FlagActSorting);
	ELSIF ManualStepAct = MANUAL_ACTUATOR_SORTING THEN
		FlagActBoth := 0;
		FlagActBothOff := NOT(FlagActBoth);
		FlagActDosing := 0;
		FlagActDosingOff := NOT(FlagActDosing);
		FlagActNone := 0;
		FlagActNoneOff := NOT(FlagActNone);
		FlagActSorting := 1;
		FlagActSortingOff := NOT(FlagActSorting);
	ELSIF ManualStepAct = MANUAL_ACTUATOR_BOTH THEN
		FlagActBoth := 1;
		FlagActBothOff := NOT(FlagActBoth);
		FlagActDosing := 1;
		FlagActDosingOff := NOT(FlagActDosing);
		FlagActNone := 0;
		FlagActNoneOff := NOT(FlagActNone);
		FlagActSorting := 1;
		FlagActSortingOff := NOT(FlagActSorting);
	ELSIF ManualStepAct = MANUAL_ACTUATOR_NONE THEN
		FlagActBoth := 0;
		FlagActBothOff := NOT(FlagActBoth);
		FlagActDosing := 0;
		FlagActDosingOff := NOT(FlagActDosing);
		FlagActNone := 1;
		FlagActNoneOff := NOT(FlagActNone);
		FlagActSorting := 0;
		FlagActSortingOff := NOT(FlagActSorting);
	END_IF;

	IF (((gMotorBeltParType.Distance < 0) AND gMotorBeltAxisBasic.MoveActive AND FlagAdd) OR ((gMotorBeltParType.Velocity <0) AND gMotorBeltAxisBasic.MoveActive AND FlagVel)) THEN
		FlagArrowLeft := 1;
		FlagArrowRight := 0;
	ELSIF (((gMotorBeltParType.Distance > 0) AND gMotorBeltAxisBasic.MoveActive AND FlagAdd) OR ((gMotorBeltParType.Velocity > 0) AND gMotorBeltAxisBasic.MoveActive AND FlagVel)) THEN
		FlagArrowRight := 1;
		FlagArrowLeft := 0;
	ELSE
		FlagArrowRight := 0;
		FlagArrowLeft := 0;
	END_IF;

	//----------------------END---OF---FLAG---SECTION----------------------------//

END_PROGRAM

PROGRAM _EXIT

END_PROGRAM
```

### Program Logical/Programs/Program (IEC)

#### Types.typ
```iecst
TYPE
	ProgramStatesEnum :
		(
		STOP,
		INIT,
		DETECTION,
		CATEGORIZATION,
		SORT_STORAGE_LEFT,
		SORT_STORAGE_RIGHT,
		SORT_WEIGHT,
		SORT_WEIGHT_AND_OPTIC,
		SORT_OPTIC,
		STOP_AND_MANUAL,
		GO_STORAGE_LEFT,
		GO_STORAGE_RIGHT,
		TAKE_PICT_CAMERA,
		DROP,
		UNRECOGNISED_PIC
	);
	SortChoiceEnum :
		(
		WEIGHT,
		WEIGHT_AND_OPTIC,
		OPTIC
	);
END_TYPE
```

#### Variables.var
```iecst
VAR
	Approval : BOOL;
	ActuatorByte : INT := 2#0000000000000000;
	ActuatorPushing : BOOL := FALSE;
	ActuatorSorting : BOOL := FALSE;
	ItemDetected : BOOL := FALSE;
	ItemWeight : USINT;
	ItemWeightChoosen : USINT := 12;
	ItemWeightMeasured : USINT;
	MotorAcc : UINT := 700;
	MotorDec : UINT := 700;
	MotorHome : BOOL;
	MotorDist : UINT := 10;
	MotorInPosition : BOOL;
	MotorMoveAbsolute : BOOL := FALSE;
	MotorMoveDone : BOOL;
	MotorPower : BOOL := FALSE;
	MotorResetError : BOOL := FALSE;
	QuantityRightStorage : UINT;
	QuantityLeftStorage : UINT;
END_VAR
VAR CONSTANT
	RESET_ITEM_MEM_WEIGHT : USINT := 0;
END_VAR
VAR
	MotorVel : {REDUND_UNREPLICABLE} UINT := 300;
	SortChoice : SortChoiceEnum := WEIGHT;
	Start : BOOL := FALSE;
	State : ProgramStatesEnum := INIT;
	Stop : BOOL := FALSE;
	TimerTonActuator : TON;
	TimerTonActuatorIn : BOOL := FALSE;
	TimerActuatorOut : BOOL;
END_VAR
VAR CONSTANT
	TIME_TON_ACTUATOR : TIME := T#500MS;
	ACTUATOR_BYTE_PUSH : INT := 2#0000000000000100;
	ACTUATOR_BYTE_SORT : INT := 2#0000000000000001;
	ACTUATOR_BYTE_NOT_ACTIV : USINT := 2#0000000000000000;
END_VAR
VAR
	MOTOR_DIST_LEFT : {REDUND_UNREPLICABLE} UINT := 90;
	MOTOR_DIST_RIGHT : {REDUND_UNREPLICABLE} UINT := 320;
	AddToLeft : BOOL;
	AddToRight : BOOL;
	CTU_QuantityLeft : CTU;
	CTU_QuantityRight : CTU;
	StringState : STRING[80];
	StringRecognisedModel : STRING[80];
	TimerCameraPicDone : BOOL;
	TimerTonCamera : TON;
END_VAR
VAR CONSTANT
	TIME_TON_CAMERA : TIME := T#4S;
END_VAR
VAR
	CTU_Reset_Left : BOOL;
	CTU_Reset_Right : BOOL;
	TimerTonDetect : TON;
	TIME_TON_DETECT : TIME := T#2S;
	TimerAfterDetect : BOOL;
	ActuatorNotSorting : BOOL;
	ActuatorNotPushing : BOOL;
	MotorReqPosition : UINT := 0;
	ErrorMaxL : BOOL;
	ErrorMaxR : BOOL;
END_VAR
```

#### Main.st
```iecst
// ALREADY WORKING, ONLY SOME CHANGES REQUIRED
PROGRAM _INIT
//	// NEED ONLY FOR WATCH
//	gAxis_1;
//	gMotorBeltParType;
//	gMotorBeltAxisBasic;
//
END_PROGRAM

PROGRAM _CYCLIC
//
//	// MOTOR MANAGEMENT
//	gMotorBeltAxisBasic.Enable 		:= TRUE;
//	gMotorBeltAxisBasic.MpLink 		:= ADR(gAxis_1);
//	gMotorBeltAxisBasic.Parameters 	:= ADR(gMotorBeltParType);
//	MotorMoveDone 					:= gMotorBeltAxisBasic.MoveDone;
//	gMotorBeltAxisBasic.Power 		:= MotorPower;
//	gMotorBeltAxisBasic.Home 		:= MotorHome;
//	// ASSIGNING MOTION PARAMETERS
//	gMotorBeltParType.Acceleration 	:= MotorAcc;
//	gMotorBeltParType.Deceleration 	:= MotorDec;
//	gMotorBeltParType.Velocity 		:= MotorVel;
//	gMotorBeltParType.Position 		:= MotorReqPosition;
//
//	gMotorBeltAxisBasic();
//
//	// ASSIGNING GLOBAL VARIABLES TO LOCAL VARIABLES
//	gActuatorByte					 := ActuatorByte;
//	gMotorBeltAxisBasic.Power 		 := MotorPower;
//	gMotorBeltAxisBasic.MoveAbsolute := MotorMoveAbsolute;
//	gMotorBeltAxisBasic.ErrorReset	 := MotorResetError;
//	// ASSIGNING LOCAL VARIABLES TO GLOBAL VARIABLES
//	MotorInPosition 				 := gMotorBeltAxisBasic.InPosition;
//	ItemDetected					 := gWeightDetected;
//	ItemWeight 						 := gInWeightMeasure;
//
//	// ITEM DETECTION CONDITION
//	ItemDetected := (ItemWeight > 1);
//
//	// TIMERS
//	// actuator
//	TimerTonActuator(IN := TimerTonActuatorIn, PT := TIME_TON_ACTUATOR);
//	TimerActuatorOut := TimerTonActuator.Q;
//	// camera
//	TimerTonCamera(IN := gImageAcq , PT := TIME_TON_CAMERA);
//	TimerCameraPicDone := TimerTonCamera.Q;
//	// delay after detection
//	TimerTonDetect.IN := ItemDetected;
//	TimerTonDetect.PT := TIME_TON_DETECT;
//	TimerAfterDetect := TimerTonDetect.Q;
//	TimerTonDetect();
//
//
//	// COUNTERS
//	CTU_QuantityLeft(CU := AddToLeft, RESET := CTU_Reset_Left, PV := gMaxLeftStorage);
//	CTU_QuantityRight(CU := AddToRight, RESET := CTU_Reset_Right, PV := gMaxRightStorage);
//	QuantityLeftStorage  := CTU_QuantityLeft.CV;
//	QuantityRightStorage := CTU_QuantityRight.CV;
//
//	//COUNTERS ALARMS (MOZE PRZERZUC DO ALARMÓW)
//	IF QuantityLeftStorage >= gMaxLeftStorage THEN
//		ErrorMaxL;
//	END_IF;
//
//	IF QuantityRightStorage >= gMaxRightStorage THEN
//		ErrorMaxR;
//	END_IF;
//
//	// PROGRAM MANUAL TURNED ON
//	IF Stop OR gMode = 1 THEN
//		Stop := FALSE;
//		State := STOP;
//	END_IF;
//	// PROGRAM AUTO
//	CASE State OF
//		STOP:
//			StringState := 'Stop';
//			IF gMode = 0 THEN
//				MotorPower := FALSE;
//				MotorMoveAbsolute := FALSE;
//				MotorHome := FALSE;
//			END_IF;
//			TimerTonActuatorIn := FALSE;
//			ActuatorSorting := FALSE;
//			ActuatorPushing := FALSE;
//			ItemWeightMeasured := RESET_ITEM_MEM_WEIGHT;
//			IF Start THEN
//				State := INIT;
//			END_IF;
//
//		INIT:
//			//Power???
//			StringState 		:= 'Inicjalizacja';
//			ItemWeightMeasured 	:= RESET_ITEM_MEM_WEIGHT;
//			AddToRight 			:= FALSE;
//			AddToLeft 			:= FALSE;
//			TimerTonActuatorIn 	:= FALSE;
//			ActuatorSorting 	:= FALSE;
//			ActuatorPushing 	:= FALSE;
//			MotorMoveAbsolute 	:= FALSE;
//			MotorPower 			:= TRUE;
//			MotorHome 			:= TRUE;
//			IF ItemDetected THEN
//				State := DETECTION;
//			END_IF;
//
//		DETECTION:
//			MotorHome 			:= FALSE;
//			StringState := 'Wykrycie detalu';
//			IF TimerAfterDetect AND Approval THEN
//				Approval := 0;
//				ItemWeightMeasured := ItemWeight;
//				State := CATEGORIZATION;
//			END_IF;
//
//		CATEGORIZATION:
//			StringState := 'Kategoryzacja detalu';
//			IF SortChoice = WEIGHT AND Approval THEN
//				Approval := 0;
//				State := DROP;
//			ELSIF SortChoice = OPTIC THEN
//				State := TAKE_PICT_CAMERA;
//			END_IF;
//
//		TAKE_PICT_CAMERA:
//			StringState := 'Robienie zdjęcia i rozpoznawanie';
//			gImageAcq 	:= TRUE; //zrob zdj na zboczu narastajacym
//			IF TimerCameraPicDone AND Approval THEN
//				Approval := 0;
//				gImageAcq := FALSE;
//				State := DROP;
//			END_IF;
//
//		DROP:
//			StringState := 'Dozowanie detalu';
//			ActuatorPushing := TRUE;
//			IF TimerActuatorOut THEN
//				ActuatorPushing := FALSE;
//				IF SortChoice = OPTIC THEN
//					State := SORT_OPTIC;
//				ELSIF SortChoice = WEIGHT THEN
//					State := SORT_WEIGHT;
//				END_IF;
//			END_IF;
//
//			// ABOVE 1 TO ItemWeightChoosen ITEM FALL INTO THE LEFT, AND ABOVE ItemWeightChoosen INTO THE RIGHT
//		SORT_WEIGHT:
//			StringState := 'Sortowanie wagowe';
//			IF ItemWeightMeasured > 1 AND ItemWeightMeasured < ItemWeightChoosen AND Approval THEN
//				Approval := 0;
//				State := GO_STORAGE_LEFT;
//			ELSIF ItemWeightMeasured >= ItemWeightChoosen AND Approval THEN
//				Approval := 0;
//				State := GO_STORAGE_RIGHT;
//			END_IF;
//
//		SORT_OPTIC:
//			StringState := 'Sortowanie optyczne';
//			IF gRecognisedModel = 0 AND Approval THEN
//				Approval := 0;
//				gImageAcq 			  := FALSE;
//				StringRecognisedModel := 'Unrecognised';
//				State 				  := UNRECOGNISED_PIC;
//			ELSIF gRecognisedModel = 1 AND Approval THEN
//				Approval := 0;
//				gImageAcq 			  := FALSE;
//				StringRecognisedModel := 'B&R';
//				State 				  := GO_STORAGE_LEFT;
//
//			ELSIF gRecognisedModel = 2 AND Approval THEN
//				Approval := 0;
//				gImageAcq 			  := FALSE;
//				StringRecognisedModel := 'AS';
//				State 			 	  := GO_STORAGE_RIGHT;
//			END_IF;
//
//		GO_STORAGE_LEFT:
//			StringState := 'Transport detalu do lewego zbiornika';
//			MotorReqPosition := MOTOR_DIST_LEFT;
//			MotorMoveAbsolute := TRUE;
//			IF MotorInPosition AND MotorMoveDone AND Approval THEN
//				Approval := 0;
//				State := SORT_STORAGE_LEFT;
//			END_IF;
//
//		GO_STORAGE_RIGHT:
//			StringState := 'Transport detalu do prawego zbiornika';
//			MotorReqPosition := MOTOR_DIST_RIGHT;
//			MotorMoveAbsolute := TRUE;
//			IF MotorInPosition AND MotorMoveDone AND Approval THEN
//				Approval := 0;
//				State := SORT_STORAGE_RIGHT;
//			END_IF;
//
//		SORT_STORAGE_LEFT:
//			StringState := 'Zepchniecie detalu z taśmy do zbiornika lewego';
//			MotorMoveAbsolute := FALSE;
//			ActuatorSorting := TRUE;
//			AddToLeft := TRUE;
//			IF TimerActuatorOut AND Approval THEN
//				Approval := 0;
//				State := INIT;
//			END_IF;
//
//		SORT_STORAGE_RIGHT:
//			AddToRight := TRUE;
//			MotorMoveAbsolute := FALSE;
//			State := INIT;
//
//		UNRECOGNISED_PIC:
//			StringState := 'Nie rozpoznano zdjęcia';
//			State := STOP;
//
//	END_CASE;
//
//
//	// TIMER INPUT TRIGGER TO DELAY ACTUATORS
//	IF ActuatorPushing OR ActuatorSorting THEN
//		TimerTonActuatorIn := TRUE;
//	ELSE
//		TimerTonActuatorIn := FALSE;
//	END_IF;
//
//	// OPERATION OF BYTE ACTUATORS WITH TIMER
//	IF ActuatorPushing THEN
//		ActuatorByte := ACTUATOR_BYTE_PUSH;
//		IF TimerActuatorOut THEN
//			ActuatorPushing := FALSE;
//		END_IF;
//	ELSIF ActuatorSorting THEN
//		ActuatorByte := ACTUATOR_BYTE_SORT;
//		IF TimerActuatorOut THEN
//			ActuatorSorting := FALSE;
//		END_IF;
//	ELSE
//		ActuatorByte := ACTUATOR_BYTE_NOT_ACTIV;
//	END_IF;
//
//	ActuatorNotSorting := NOT ActuatorSorting;
//	ActuatorNotPushing 	:= NOT ActuatorPushing;
//
//	IF Start THEN
//		Start := FALSE;
//	END_IF;
//
				END_PROGRAM

PROGRAM _EXIT

				END_PROGRAM
```

### Program Logical/Programs/RecipesMgmnt (IEC)

#### Variables.var
```iecst
VAR
	lol : USINT;
END_VAR
```

#### Main.st
```iecst
PROGRAM _INIT
	(* Insert code here *)

END_PROGRAM

PROGRAM _CYCLIC
	//FileName := 'elo';

	gMpRecipeXML_0.MpLink := 		ADR(gRecipeXml);
	gMpRecipeXML_0.Enable := 		TRUE;
	gMpRecipeXML_0.DeviceName :=	ADR('CF');
	gMpRecipeXML_0.FileName := 		ADR('FileNameEee'); //zmienic sciezke

	gMpRecipeRegPar_0.MpLink := 	ADR(gRecipeXml);
	gMpRecipeRegPar_0.Enable :=		TRUE;
	gMpRecipeRegPar_0.PVName := 	ADR('gSorting');

	gMpRecipeUI_0.MpLink :=			ADR(gRecipeXml);
	gMpRecipeUI_0.Enable := 		TRUE;
	gMpRecipeUI_0.UISetup := 		gUISetup;
	gMpRecipeUI_0.UIConnect := 		ADR(gUIConnect);

	gSorting.ItemWeightChoosen;
	gSorting.RecognisedModel; //CO TU DAC???
	gSorting.SortLeftMin;
	gSorting.SortChoice;

	//	Parametry sortowania powinno dac sie zapisac oraz wczytac przy uzyciu systemu receptur
	//	MpRecipe. Na stronie parametrów powinna wiec istniec mozliwosc przegladania listy dostepnych receptur,
	//	wczytania receptury z listy, zapisania nowej receptury oraz modyfikacji parametrów dowolnej z zapisanych
	//	receptur. Powinno byc takze mozliwe wyswietlenie parametrów danej receptury bez wczytywania jej oraz
	//	calkowite usuniecie receptury widocznej na liscie. Zarówno na stronie parametrów jak i na stronie pracy automatycznej (oraz przy pracy pólautomatycznej) powinna byc wyswietlona obecnie wczytana receptura,
	//	chyba ze uzywane sa aktualnie niezapisane DO receptury, recznie ustawione, parametry sortowania.

	gMpRecipeUI_0();
	gMpRecipeXML_0();
	gMpRecipeRegPar_0();
END_PROGRAM

PROGRAM _EXIT
	(* Insert code here *)

END_PROGRAM
```

### Program Logical/Programs/Camera (IEC)

#### Variables.var
```iecst
VAR
	ATON1 : TON;
	ATON2 : TON;
	ATON3 : TON;
	Base64Buffer : STRING[2500000];
	Base64srcLen : UDINT;
	CameraLED : USINT := 0;
	CameraLED_2 : USINT := 0;
	CameraLED_OPC : USINT := 0;
	CTU_HowManyBlink : CTU;
	EXPO_TIME : {REDUND_UNREPLICABLE} UDINT := 15000;
	FLASH_COLOR : {REDUND_UNREPLICABLE} USINT := 1;
	FLASH_SEGMENT : {REDUND_UNREPLICABLE} USINT := 1;
	httpDecodeBase64_0 : httpDecodeBase64;
	httpEncodeBase64_0 : httpEncodeBase64;
	ImageProcess : USINT;
	ImgProcessingActive : BOOL;
END_VAR
VAR CONSTANT
	LED_BLUE : USINT := 4;
	LED_GREEN : USINT := 2;
	LED_NOTHING : USINT := 1;
	LED_PLC_STATUS : USINT := 0;
	LED_RED : USINT := 3;
END_VAR
VAR
	ManualLampTest : BOOL;
	MatchEnable : BOOL := TRUE;
	MatchScore : USINT;
	MAX_OVERLAP : USINT := 0;
	MIN_SCORE : USINT := 44;
	NewEncodeReq : BOOL;
	NumberMatches : USINT;
	NUM_SEARCH_MAX : USINT := 1;
	OneMoreBlink : BOOL;
	PhotosTaken : USINT;
	RecognisedModel : USINT;
	SET_FOCUS : UINT := 15000;
	sStep : INT;
	TestStringURL : STRING[2600000];
	TimerTonCameraLED : TON;
	TimerTonCameraLED_2 : TON;
END_VAR
VAR CONSTANT
	TIMER_TIME_BLINK : TIME := T#500MS;
	TIMER_TIME_BLINK_100MS : TIME := T#100MS;
	TIMER_TIME_BLINK_500MS : TIME := T#500MS;
	TIME_LAMP_TEST : TIME := T#500MS;
END_VAR
VAR
	URL : STRING[2600000];
	URLLength : UDINT;
	ViBaseBuffer : ARRAY[0..1500000] OF USINT := [1500001(1)];
	ViBaseGetImage_0 : ViBaseGetImage;
	VIBASE_GETIMG_QUALITY : USINT := 5;
END_VAR
```
